(* IEC 61131-3 sources: volt/packages/volt-lsp-iec/test-corpus/awa-palletizer/Device/Plc Logic/Application/140 UN01_Palletizer, 4 files *)

(* ---- UN01_GVL.gvl ---- *)
{attribute 'qualified_only'}
{attribute 'symbol' := 'none'}
VAR_GLOBAL
	//PH01_Picking : ARRAY[1..3] OF PH_Picking;
END_VAR

(* ---- UN01_HMI.gvl ---- *)
{attribute 'qualified_only'}
{attribute 'symbol' := 'readwrite'}
VAR_GLOBAL
	{attribute 'symbol' := 'readwrite'}
	EM01_PickingStation_HMI: ARRAY[1..3] OF dutPickingStation_HMI;
	{attribute 'symbol' := 'readwrite'}
	EM02_PalletPosition_HMI: ARRAY[1..4] OF dutPalletPosition_HMI;
	{attribute 'symbol' := 'readwrite'}
	EM02_PalletPositionActuals_HMI: ARRAY[1..3] OF dutPalletPositionActuals_HMI;
	{attribute 'symbol' := 'readwrite'}
	EM02_CoordSystem_HMI: ARRAY[1..12] OF dutCoordSystem_HMI;
	{attribute 'symbol' := 'readwrite'}
	EM02_PalletizerControl_HMI: dutPalletizerControl_HMI;
	{attribute 'symbol' := 'readwrite'}
	RecipeView_HMI: dutRecipeView_HMI;
	{attribute 'symbol' := 'readwrite'}
	RecipeSelect_HMI: dutRecipeSelect_HMI;
	{attribute 'symbol' := 'readwrite'}
	CoordSystemOffset_HMI: dutCoordSystemOffset_HMI;
	{attribute 'symbol' := 'readwrite'}
	UN01_HMI: dutHMI;
	{attribute 'symbol' := 'readwrite'}
	iTest:INT;
END_VAR

(* ---- UN01_IO.gvl ---- *)
{attribute 'qualified_only'}
VAR_GLOBAL
	// Conveyor 1
	QxMOT01_Conveyor: BOOL := FALSE;
	// Conveyor 2
	QxMOT02_Conveyor: BOOL := FALSE;
	// Conveyor 3
	QxMOT03_Conveyor: BOOL := FALSE;

	// Conveyor 1
	IxMOT01_ThermOk: BOOL := FALSE;
	// Conveyor 2
	IxMOT02_ThermOk: BOOL := FALSE;
	// Conveyor 3
	IxMOT03_ThermOk: BOOL := FALSE;
	// Box at position
	IxSEN01_Box01: BOOL := FALSE;
	// Box at position
	IxSEN01_Box02: BOOL := FALSE;
	// Box at position
	IxSEN01_Box03: BOOL := FALSE;
	// Box at position
	IxSEN01_Box04: BOOL := FALSE;
	// Box at position
	IxSEN02_Box01: BOOL := FALSE;
	// Box at position
	IxSEN02_Box02: BOOL := FALSE;
	// Box at position
	IxSEN02_Box03: BOOL := FALSE;
	// Box at position
	IxSEN02_Box04: BOOL := FALSE;
	// Box at position
	IxSEN03_Box01: BOOL := FALSE;
	// Box at position
	IxSEN03_Box02: BOOL := FALSE;
	// Box at position
	IxSEN03_Box03: BOOL := FALSE;
	// Box at position
	IxSEN03_Box04: BOOL := FALSE;
	// Request box
	QxDO01_InputEnable: BOOL := FALSE;
	// Request box
	QxDO02_InputEnable: BOOL := FALSE;
	// Request box
	QxDO03_InputEnable: BOOL := FALSE;
END_VAR

(* ---- UN01_Main.pou ---- *)
FUNCTION_BLOCK UN01_Main EXTENDS StateMachine;
VAR
	myState 		: strState;			// Unit state
	iIndex			: INT;
END_VAR

%LANGUAGE ST
{region}

	{region}

	//----------------------------------------------------------------------------------
	// STATE CONTROL
	//----------------------------------------------------------------------------------

		myState.xCmdInit  S= (FALSE					   );
		myState.xCmdReset S= (PC01_GVL.BTN03_Reset.xDI );
		myState.xCmdStart S= (PC01_GVL.BTN01_Start.xDI );
		myState.xCmdStop  S= (PC01_GVL.BTN02_Stop.xDI  );
		myState.xCmdAbort S= (FALSE					   );

		SUPER^.Handle(_HMI := UN01_HMI.UN01_HMI, myState := myState);
	{endregion}

	//CONTROL MODULES
	{region}

		xCMError	:= FALSE;

		//---------------------------------------------------------------------------------------------
		// Control Modules.
		//---------------------------------------------------------------------------------------------

		//---------------------------------------------------------------------------------------------
		// Phase Modules.
		//---------------------------------------------------------------------------------------------
{*
		FOR iIndex := 1 TO 3 DO
			UN01_GVL.PH01_Picking[iIndex](
				PickingStation:= UN01_GVL.EM01_PickingStation[iIndex],
				SFCInit:= myState.xStsInit,
				SFCReset:= myState.xStsResetting,
				SFCExecute:= myState.xStsExecute,
				SFCPause:= NOT(myState.xStsExecute),
				SFCAbort:= myState.xStsAborting OR myState.xStsAborted,
				SFCError=> ,
				xStsReadyForPick=> ,
				xStsFull=>,
				IQ_ModuleHandler := myModuleHandler );
		END_FOR
*}
		//---------------------------------------------------------------------------------------------
		// Always!
		//---------------------------------------------------------------------------------------------

	{endregion}

	//ALARM
	{region}
		myState.xCmdAbort := xCMError;

		// For debugging purposes.
		IF (myState.xCmdAbort) THEN
			myState.xCmdAbort := true;
		END_IF
	{endregion}
{endregion}

{region}
	//------------------------------------------------------------------------------------------------------
	// Alarm and warning handling.
	//------------------------------------------------------------------------------------------------------

	wErrorID := 16#0000;
	wWarningID := 16#0000;

	//Alarm
	ALM_Error(
		ModuleHandler:= myModuleHandler,
		ErrorHandler:= ,
		xSetError:= (wErrorID <> 0),
		eSeverity:= L_IE1P.L_IE1P_SeverityLevel.Fault,
		wTextRefId:= GVL_Errorlists.PC01_TextList,
		wErrorId:= wErrorID,
		eReaction:= L_IE1P.L_IE1P_Reaction.NormalStop);

	//Warning
	ALM_Warning(
		ModuleHandler:= myModuleHandler,
		ErrorHandler:= ,
		xSetError:= (wWarningID <> 0),
		eSeverity:= L_IE1P.L_IE1P_SeverityLevel.Warning,
		wTextRefId:= GVL_Errorlists.PC01_TextList,
		wErrorId:= wWarningID,
		eReaction:= L_IE1P.L_IE1P_Reaction.No_Reaction);

	IF NOT xInitProgramAlarms THEN
		myModuleHandler.SetParent(ModuleHandlerParent:= myModuleHandler);
		xInitProgramAlarms:= TRUE;
	END_IF

	ForwardAlarms(
		xEnable:= TRUE,
		ModuleHandler:= myModuleHandler,
		xForwardFromChildModules:=TRUE);
{endregion}

END_FUNCTION_BLOCK

ACTION Aborted
%LANGUAGE ST
//----------------------------------------------------------------------------------
// Aborted
//----------------------------------------------------------------------------------

END_ACTION

ACTION Aborting
%LANGUAGE ST
//----------------------------------------------------------------------------------
// Aborting
//----------------------------------------------------------------------------------

myState.xCmdAbortDone := TRUE;
END_ACTION

ACTION Executing
%LANGUAGE ST
//-------------------------------------------------------------------------------------
// Executing
//-------------------------------------------------------------------------------------

END_ACTION

ACTION Idle
%LANGUAGE ST
//-------------------------------------------------------------------------------------
// Idle
//-------------------------------------------------------------------------------------

END_ACTION

ACTION Initialize
%LANGUAGE ST
//-------------------------------------------------------------------------------------
// Initialize
//-------------------------------------------------------------------------------------

UN01_HMI.EM02_CoordSystem_HMI[1].iCoordSystemId := 1;
UN01_HMI.EM02_CoordSystem_HMI[1].strName := 'Picking 1';

UN01_HMI.EM02_CoordSystem_HMI[2].iCoordSystemId := 2;
UN01_HMI.EM02_CoordSystem_HMI[2].strName := 'Picking 2';

UN01_HMI.EM02_CoordSystem_HMI[3].iCoordSystemId := 3;
UN01_HMI.EM02_CoordSystem_HMI[3].strName := 'Picking 3';

UN01_HMI.EM02_CoordSystem_HMI[4].iCoordSystemId := 4;
UN01_HMI.EM02_CoordSystem_HMI[4].strName := 'WCS';

UN01_HMI.EM02_CoordSystem_HMI[5].iCoordSystemId := 5;
UN01_HMI.EM02_CoordSystem_HMI[5].strName := 'Pallet 1';

UN01_HMI.EM02_CoordSystem_HMI[6].iCoordSystemId := 6;
UN01_HMI.EM02_CoordSystem_HMI[6].strName := 'Pallet 2';

UN01_HMI.EM02_CoordSystem_HMI[7].iCoordSystemId := 7;
UN01_HMI.EM02_CoordSystem_HMI[7].strName := 'Pallet 3';

UN01_HMI.EM02_CoordSystem_HMI[8].iCoordSystemId := 8;
UN01_HMI.EM02_CoordSystem_HMI[8].strName := 'IML 1';

UN01_HMI.EM02_CoordSystem_HMI[9].iCoordSystemId := 9;
UN01_HMI.EM02_CoordSystem_HMI[9].strName := 'IML 2';

UN01_HMI.EM02_CoordSystem_HMI[10].iCoordSystemId := 10;
UN01_HMI.EM02_CoordSystem_HMI[10].strName := 'IML 3';

UN01_HMI.EM02_CoordSystem_HMI[11].iCoordSystemId := 11;
UN01_HMI.EM02_CoordSystem_HMI[11].strName := 'IML 4';

UN01_HMI.EM02_CoordSystem_HMI[12].iCoordSystemId := 12;
UN01_HMI.EM02_CoordSystem_HMI[12].strName := 'Home';

UN01_HMI.EM01_PickingStation_HMI[1].iStation := 1;
UN01_HMI.EM01_PickingStation_HMI[1].strName := 'Picking 1';

UN01_HMI.EM01_PickingStation_HMI[2].iStation := 2;
UN01_HMI.EM01_PickingStation_HMI[2].strName := 'Picking 2';

UN01_HMI.EM01_PickingStation_HMI[3].iStation := 3;
UN01_HMI.EM01_PickingStation_HMI[3].strName := 'Picking 3';

UN01_HMI.EM02_PalletPositionActuals_HMI[1].iPalletPositionNr := 1;
UN01_HMI.EM02_PalletPositionActuals_HMI[1].strName := 'Pallet 1';

UN01_HMI.EM02_PalletPositionActuals_HMI[2].iPalletPositionNr := 2;
UN01_HMI.EM02_PalletPositionActuals_HMI[2].strName := 'Pallet 2';

UN01_HMI.EM02_PalletPositionActuals_HMI[3].iPalletPositionNr := 3;
UN01_HMI.EM02_PalletPositionActuals_HMI[3].strName := 'Pallet 3';

END_ACTION

ACTION Resetting
%LANGUAGE ST
//-------------------------------------------------------------------------------------
// Resetting
//-------------------------------------------------------------------------------------

UN01_HMI.RecipeSelect_HMI.iPalletPositionId := 0;
UN01_HMI.RecipeView_HMI.iPalletPositionId := 0;
UN01_HMI.CoordSystemOffset_HMI.iCoordSystemId := 1;

myState.xCmdResetDone := TRUE;
END_ACTION

ACTION Starting
%LANGUAGE ST
//-------------------------------------------------------------------------------------
// Starting
//-------------------------------------------------------------------------------------

myState.xCmdStartDone := TRUE;
END_ACTION

ACTION Stopped
%LANGUAGE ST
//-------------------------------------------------------------------------------------
// Stopped
//-------------------------------------------------------------------------------------

END_ACTION

ACTION Stopping
%LANGUAGE ST
//-------------------------------------------------------------------------------------
// Stopping
//-------------------------------------------------------------------------------------

myState.xCmdStopDone := TRUE;
END_ACTION
